{attribute 'GeneratedUsingTerminal: EJ1914-0000-0017'}
{attribute addProperty BoxType "EJ1914-0000-0017"}
{attribute addProperty Id "FSOEAT %I*FSOE_1F44E1B411"}
{attribute addProperty CRC "2303917808"}
{attribute addProperty Size "11"}
TYPE FSoE_Inputs_8952FEF0 EXTENDS InputBase_8311D824 :
STRUCT
	{attribute addProperty Name "FSOE"}
	FSOE AT %I* : FSOE_1F44E1B4;
END_STRUCT
END_TYPE

(* stored: Version 1.2.0.0, ProductVersion 3.1.4024.9
   DUT FSoE_Inputs_8952FEF0: Id {1c9f6a77-8432-4e6f-a7d6-35a94042a2f1} *)
